PROGRAM IP232
VAR
	timer				: TON;
	bDoReading			: BOOL;
	
	bOnInit				: BOOL	:= TRUE;
	timerInit			: TON;
	
	nState				: INT;
	
	fbInit232_01_5350			: FB_InitPM;
	fbInit232_03_5350			: FB_InitPM;
	fbInit232_05_5350			: FB_InitPM;
	fbInit232_07_5350			: FB_InitPM;
	fbInit232_08_5350			: FB_InitPM;
	
	fbRead232_01_5350			: FB_ReadPM5350;
	fbRead232_03_5350			: FB_ReadPM5350;
	fbRead232_05_5350			: FB_ReadPM5350;
	fbRead232_07_5350			: FB_ReadPM5350;
	fbRead232_08_5350			: FB_ReadPM5350;
	
	fbInit232_02_5500			: FB_InitPM;
	fbInit232_04_5500			: FB_InitPM;
	fbInit232_06_5500			: FB_InitPM;
	
	fbRead232_02_5500			: FB_ReadPM5500;
	fbRead232_04_5500			: FB_ReadPM5500;
	fbRead232_06_5500			: FB_ReadPM5500;
	
	nCount						: DINT;
END_VAR

VAR CONSTANT
	STATE_INIT			:	INT		:= 0;
	STATE_READ1			:	INT		:= 10;
	STATE_READ3			:	INT		:= 30;
	STATE_READ5			:	INT		:= 50;
	STATE_READ7			:	INT		:= 70;
	STATE_READ8			:	INT		:= 80;
	STATE_READ2			:	INT		:= 20;
	STATE_READ4			:	INT		:= 40;
	STATE_READ6			:	INT		:= 60;
END_VAR

timerInit(In:=TRUE, PT:=T#3S);
IF timerInit.Q THEN
	timerInit(In:=FALSE);
		bOnInit	:= FALSE;
	END_IF

IF bOnInit THEN
	fbInit232_01_5350(	sIpAddress	:= '10.91.37.232',
						nPort		:= 502,
						nUnitID		:= 1,
						PM			:= pmDev.DB02_01_5350);
	fbInit232_03_5350(	sIpAddress	:= '10.91.37.232',
						nPort		:= 502,
						nUnitID		:= 3,
						PM			:= pmDev.DB02_03_5350);
	fbInit232_05_5350(	sIpAddress	:= '10.91.37.232',
						nPort		:= 502,
						nUnitID		:= 5,
						PM			:= pmDev.DB02_05_5350);
	fbInit232_07_5350(	sIpAddress	:= '10.91.37.232',
						nPort		:= 502,
						nUnitID		:= 7,
						PM			:= pmDev.DB02_07_5350);
	fbInit232_08_5350(	sIpAddress	:= '10.91.37.232',
						nPort		:= 502,
						nUnitID		:= 8,
						PM			:= pmDev.DB02_08_5350);
						
	fbInit232_02_5500(	sIpAddress	:= '10.91.37.232',
						nPort		:= 502,
						nUnitID		:= 2,
						PM			:= pmDev.DB02_02_5500);
	fbInit232_04_5500(	sIpAddress	:= '10.91.37.232',
						nPort		:= 502,
						nUnitID		:= 4,
						PM			:= pmDev.DB02_04_5500);
	fbInit232_06_5500(	sIpAddress	:= '10.91.37.232',
						nPort		:= 502,
						nUnitID		:= 6,
						PM			:= pmDev.DB02_06_5500);
END_IF

IF NOT bOnInit THEN
	timer(In:=TRUE, PT:=T#5M);
	IF timer.Q OR pmdev.bTrigReadCOmmision THEN
		timer(In:=FALSE);
		nState	:= STATE_READ1;
	END_IF
END_IF

CASE nState OF
STATE_INIT:
	nCount	:= nCount + 1;
STATE_READ1:
	fbRead232_01_5350(
		bExecute:=TRUE,
		PM:= pmDev.DB02_01_5350);
	IF NOT fbRead232_01_5350.Q THEN
		nState	:= STATE_READ3;
		fbRead232_01_5350(
			bExecute:=FALSE,
			PM:= pmDev.DB02_01_5350);
	END_IF
	
STATE_READ3:
	fbRead232_03_5350(
		bExecute:=TRUE,
		PM:= pmDev.DB02_03_5350);
	IF NOT fbRead232_03_5350.Q THEN
		nState	:= STATE_READ5;
		fbRead232_03_5350(
			bExecute:=FALSE,
			PM:= pmDev.DB02_03_5350);
	END_IF	

STATE_READ5:
	fbRead232_05_5350(
		bExecute:=TRUE,
		PM:= pmDev.DB02_05_5350);
	IF NOT fbRead232_05_5350.Q THEN
		nState	:= STATE_READ7;
		fbRead232_05_5350(
			bExecute:=FALSE,
			PM:= pmDev.DB02_05_5350);
	END_IF	
	
STATE_READ7:
	fbRead232_07_5350(
		bExecute:=TRUE,
		PM:= pmDev.DB02_07_5350);
	IF NOT fbRead232_07_5350.Q THEN
		nState	:= STATE_READ8;
		fbRead232_07_5350(
			bExecute:=FALSE,
			PM:= pmDev.DB02_07_5350);
	END_IF	
	
STATE_READ8:
	fbRead232_08_5350(
		bExecute:=TRUE,
		PM:= pmDev.DB02_08_5350);
	IF NOT fbRead232_08_5350.Q THEN
		nState	:= STATE_READ2;
		fbRead232_08_5350(
			bExecute:=FALSE,
			PM:= pmDev.DB02_08_5350);
	END_IF	
	
STATE_READ2:
	fbRead232_02_5500(
		bExecute:=TRUE,
		PM:= pmDev.DB02_02_5500);
	IF NOT fbRead232_02_5500.Q THEN
		nState	:= STATE_READ4;
		fbRead232_02_5500(
			bExecute:=FALSE,
			PM:= pmDev.DB02_02_5500);
	END_IF
STATE_READ4:
	fbRead232_04_5500(
		bExecute:=TRUE,
		PM:= pmDev.DB02_04_5500);
	IF NOT fbRead232_04_5500.Q THEN
		nState	:= STATE_READ6;
		fbRead232_04_5500(
			bExecute:=FALSE,
			PM:= pmDev.DB02_04_5500);
	END_IF

STATE_READ6:
	fbRead232_06_5500(
		bExecute:=TRUE,
		PM:= pmDev.DB02_06_5500);
	IF NOT fbRead232_06_5500.Q THEN
		nState	:= STATE_INIT;
		fbRead232_06_5500(
			bExecute:=FALSE,
			PM:= pmDev.DB02_06_5500);
	END_IF
	
END_CASE

END_PROGRAM

(* stored: Version 1.1.0.1, ProductVersion 3.1.4024.12
   POU IP232: Id {37190f96-fa45-48ec-ac99-3bc64ba82a5f}, SpecialFunc None *)
